{attribute 'GeneratedUsingTerminal: EPP1518-0002-0016'}
{attribute addProperty BoxType "EPP1518-0002-0016"}
{attribute addProperty Id "Set_counter_doneBOOL1Counter_inhibitedBOOL1Status_of_input_UDBOOL1Status_of_input_clockBOOL1Sync_errorBOOL1TxPDO_StateBOOL1TxPDO_ToggleBOOL1"}
{attribute addProperty CRC "1464409585"}
{attribute addProperty Size "7"}
TYPE Status_57491DF1 :
STRUCT
	{attribute addProperty Name "Set_counter_done"}
	Set_counter_done : BOOL;
	{attribute addProperty Name "Counter_inhibited"}
	Counter_inhibited : BOOL;
	{attribute addProperty Name "Status_of_input_UD"}
	Status_of_input_UD : BOOL;
	{attribute addProperty Name "Status_of_input_clock"}
	Status_of_input_clock : BOOL;
	{attribute addProperty Name "Sync_error"}
	Sync_error : BOOL;
	{attribute addProperty Name "TxPDO_State"}
	TxPDO_State : BOOL;
	{attribute addProperty Name "TxPDO_Toggle"}
	TxPDO_Toggle : BOOL;
END_STRUCT
END_TYPE

(* stored: Version 1.2.0.0, ProductVersion 3.1.4024.11
   DUT Status_57491DF1: Id {15b7c654-aa77-460d-872f-129e48729d97} *)
